
// ===== library types =====

TYPE "typeADD"
   STRUCT
      addEnable : Bool;
      addNumber1 : Int;
      addNumber2 : Int;
      addOut : Int;
   END_STRUCT;
END_TYPE

FUNCTION_BLOCK "fbADD"   // FB100, FBD
{ S7_Optimized_Access := 'TRUE' }
VERSION : 0.1
   VAR_IN_OUT
      add : "typeADD";
   END_VAR
BEGIN

REGION Network 2 (SCL)
   IF #add.addEnable THEN
       #add.addOut := #add.addNumber1 + #add.addNumber2;
   END_IF;
END_REGION
END_FUNCTION_BLOCK

(* ===== HMI "HMI_RT_1" =====
system functions are stored by id; their names below are inferred from use

ScreenModuleEditorView "facePlate" 640x480
   Button "enableButton" at 27,41 size 96x32; TextOn 'enable'; TextOff 'enable'
      on Click: InvertBit("addType.addEnable")
   IOField "addNumber1" at 27,104 size 118x36; FormatPattern 9999999
      ProcessValue <- "addType.addNumber1"
   IOField "addNumber2" at 27,172 size 118x36; FormatPattern 9999999
      ProcessValue <- "addType.addNumber2"
   IOField "addOut" at 27,245 size 118x36; FormatPattern 9999999
      ProcessValue <- "addType.addOut"
*)